{attribute 'qualified_only'}
{attribute 'strict'}
TYPE SystemControlMode :
(
	Debug := 0,
	ConstForce := 1
);
END_TYPE

(* stored: Version 1.1.0.1, ProductVersion 3.1.4024.11
   DUT SystemControlMode: Id {7502ce60-9fc1-4346-9370-c09999097018} *)
